DATA_BLOCK "NetDb"
{ S7_Optimized_Access := 'TRUE' }
AUTHOR : Searinox
VERSION : 0.1
NON_RETAIN
"Net"

BEGIN

END_DATA_BLOCK

